FUNCTION_BLOCK DIV_SINT (* IEC 61131-3 SINT Division *)
  (* Standard: 61131-3 *)
  (* Version 0.0, 2004-12-15, JHC, Rockwell Automation, Converted from SRC format. *)
  (* Compiler header: package fb.rt.plc.math; *)
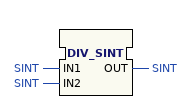
  VAR_INPUT
    IN1 : SINT; (* Dividend *)
    IN2 : SINT; (* Divisor *)
  END_VAR
  VAR_OUTPUT
    OUT : SINT; (* Quotient *)
  END_VAR
END_FUNCTION_BLOCK
